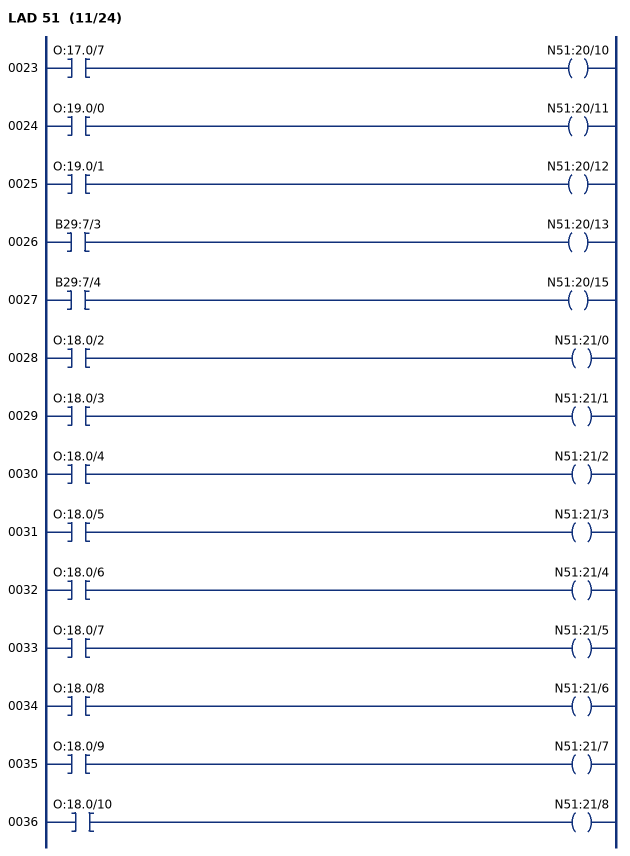
% Rung: 23 %
SOR XIC O:17.0/7 OTE N51:20/10 EOR
% Rung: 24 %
SOR XIC O:19.0/0 OTE N51:20/11 EOR
% Rung: 25 %
SOR XIC O:19.0/1 OTE N51:20/12 EOR
% Rung: 26 %
SOR XIC B29:7/3 OTE N51:20/13 EOR
% Rung: 27 %
SOR XIC B29:7/4 OTE N51:20/15 EOR
% Rung: 28 %
SOR XIC O:18.0/2 OTE N51:21/0 EOR
% Rung: 29 %
SOR XIC O:18.0/3 OTE N51:21/1 EOR
% Rung: 30 %
SOR XIC O:18.0/4 OTE N51:21/2 EOR
% Rung: 31 %
SOR XIC O:18.0/5 OTE N51:21/3 EOR
% Rung: 32 %
SOR XIC O:18.0/6 OTE N51:21/4 EOR
% Rung: 33 %
SOR XIC O:18.0/7 OTE N51:21/5 EOR
% Rung: 34 %
SOR XIC O:18.0/8 OTE N51:21/6 EOR
% Rung: 35 %
SOR XIC O:18.0/9 OTE N51:21/7 EOR
% Rung: 36 %
SOR XIC O:18.0/10 OTE N51:21/8 EOR

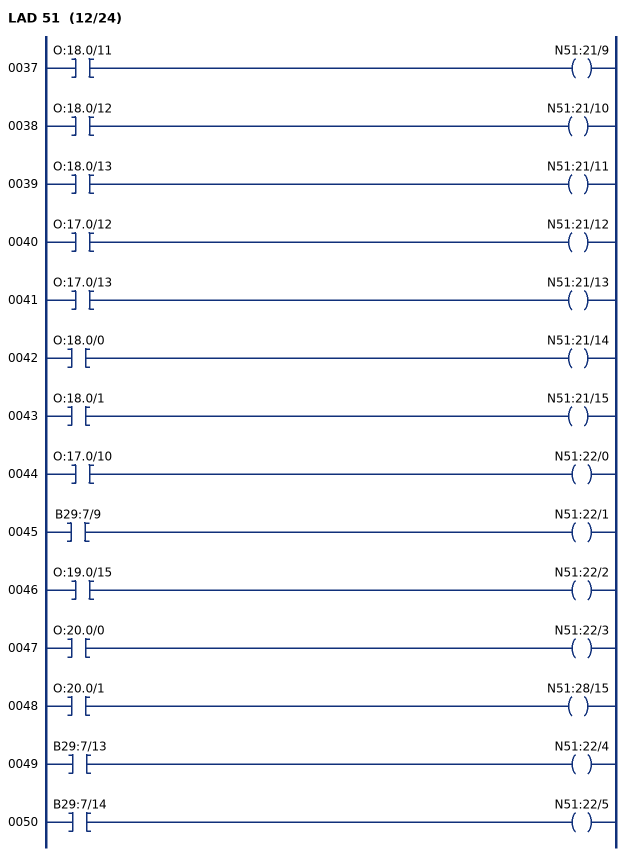
% Rung: 37 %
SOR XIC O:18.0/11 OTE N51:21/9 EOR
% Rung: 38 %
SOR XIC O:18.0/12 OTE N51:21/10 EOR
% Rung: 39 %
SOR XIC O:18.0/13 OTE N51:21/11 EOR
% Rung: 40 %
SOR XIC O:17.0/12 OTE N51:21/12 EOR
% Rung: 41 %
SOR XIC O:17.0/13 OTE N51:21/13 EOR
% Rung: 42 %
SOR XIC O:18.0/0 OTE N51:21/14 EOR
% Rung: 43 %
SOR XIC O:18.0/1 OTE N51:21/15 EOR
% Rung: 44 %
SOR XIC O:17.0/10 OTE N51:22/0 EOR
% Rung: 45 %
SOR XIC B29:7/9 OTE N51:22/1 EOR
% Rung: 46 %
SOR XIC O:19.0/15 OTE N51:22/2 EOR
% Rung: 47 %
SOR XIC O:20.0/0 OTE N51:22/3 EOR
% Rung: 48 %
SOR XIC O:20.0/1 OTE N51:28/15 EOR
% Rung: 49 %
SOR XIC B29:7/13 OTE N51:22/4 EOR
% Rung: 50 %
SOR XIC B29:7/14 OTE N51:22/5 EOR

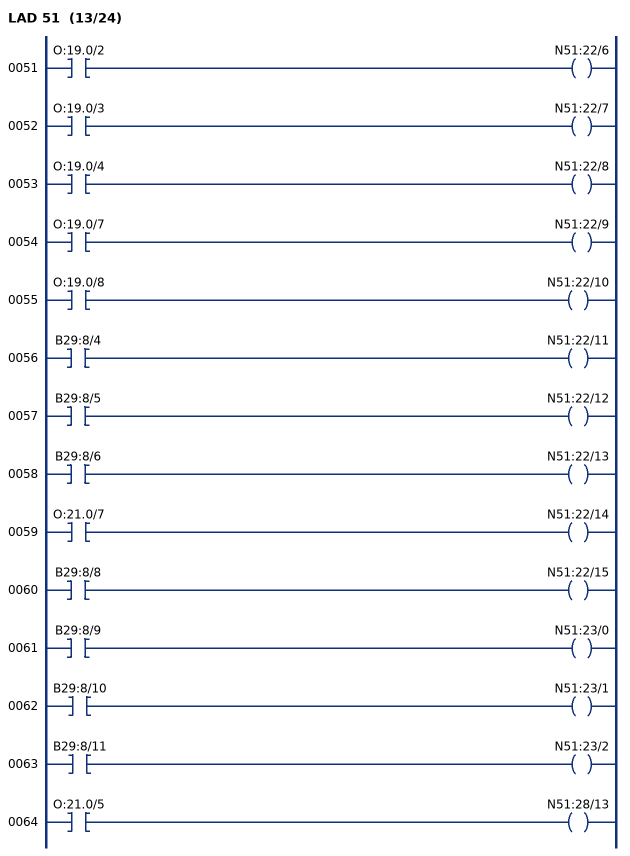
% Rung: 51 %
SOR XIC O:19.0/2 OTE N51:22/6 EOR
% Rung: 52 %
SOR XIC O:19.0/3 OTE N51:22/7 EOR
% Rung: 53 %
SOR XIC O:19.0/4 OTE N51:22/8 EOR
% Rung: 54 %
SOR XIC O:19.0/7 OTE N51:22/9 EOR
% Rung: 55 %
SOR XIC O:19.0/8 OTE N51:22/10 EOR
% Rung: 56 %
SOR XIC B29:8/4 OTE N51:22/11 EOR
% Rung: 57 %
SOR XIC B29:8/5 OTE N51:22/12 EOR
% Rung: 58 %
SOR XIC B29:8/6 OTE N51:22/13 EOR
% Rung: 59 %
SOR XIC O:21.0/7 OTE N51:22/14 EOR
% Rung: 60 %
SOR XIC B29:8/8 OTE N51:22/15 EOR
% Rung: 61 %
SOR XIC B29:8/9 OTE N51:23/0 EOR
% Rung: 62 %
SOR XIC B29:8/10 OTE N51:23/1 EOR
% Rung: 63 %
SOR XIC B29:8/11 OTE N51:23/2 EOR
% Rung: 64 %
SOR XIC O:21.0/5 OTE N51:28/13 EOR

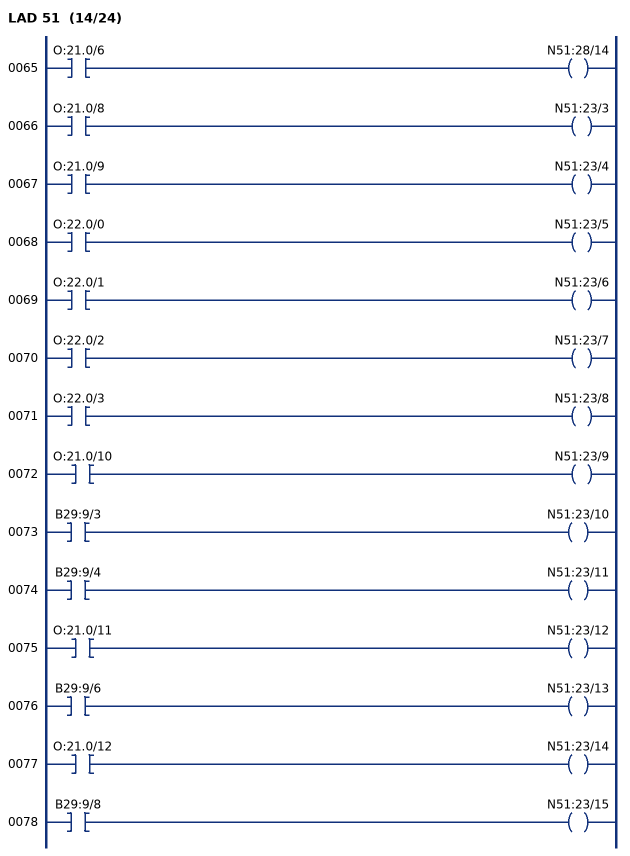
% Rung: 65 %
SOR XIC O:21.0/6 OTE N51:28/14 EOR
% Rung: 66 %
SOR XIC O:21.0/8 OTE N51:23/3 EOR
% Rung: 67 %
SOR XIC O:21.0/9 OTE N51:23/4 EOR
% Rung: 68 %
SOR XIC O:22.0/0 OTE N51:23/5 EOR
% Rung: 69 %
SOR XIC O:22.0/1 OTE N51:23/6 EOR
% Rung: 70 %
SOR XIC O:22.0/2 OTE N51:23/7 EOR
% Rung: 71 %
SOR XIC O:22.0/3 OTE N51:23/8 EOR
% Rung: 72 %
SOR XIC O:21.0/10 OTE N51:23/9 EOR
% Rung: 73 %
SOR XIC B29:9/3 OTE N51:23/10 EOR
% Rung: 74 %
SOR XIC B29:9/4 OTE N51:23/11 EOR
% Rung: 75 %
SOR XIC O:21.0/11 OTE N51:23/12 EOR
% Rung: 76 %
SOR XIC B29:9/6 OTE N51:23/13 EOR
% Rung: 77 %
SOR XIC O:21.0/12 OTE N51:23/14 EOR
% Rung: 78 %
SOR XIC B29:9/8 OTE N51:23/15 EOR

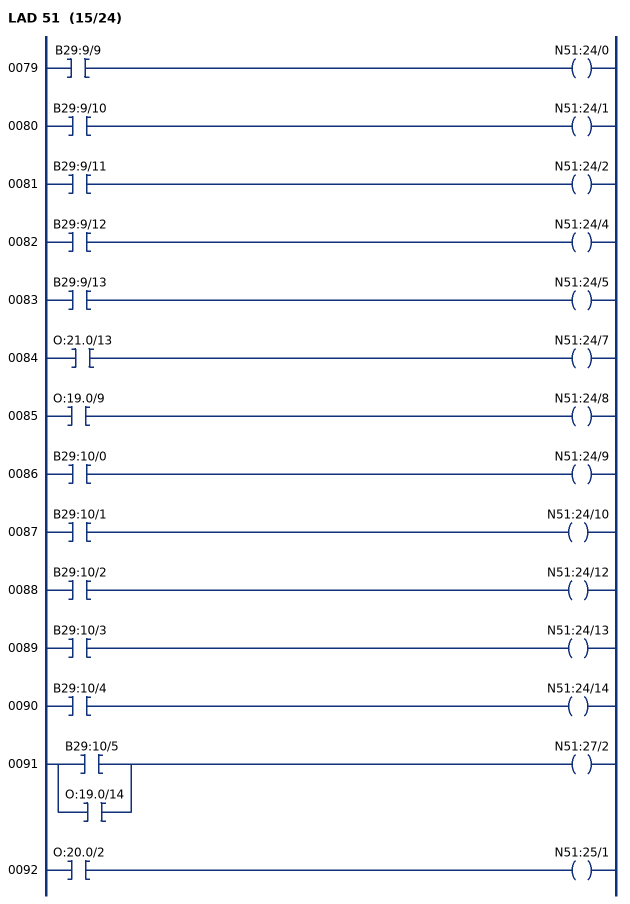
% Rung: 79 %
SOR XIC B29:9/9 OTE N51:24/0 EOR
% Rung: 80 %
SOR XIC B29:9/10 OTE N51:24/1 EOR
% Rung: 81 %
SOR XIC B29:9/11 OTE N51:24/2 EOR
% Rung: 82 %
SOR XIC B29:9/12 OTE N51:24/4 EOR
% Rung: 83 %
SOR XIC B29:9/13 OTE N51:24/5 EOR
% Rung: 84 %
SOR XIC O:21.0/13 OTE N51:24/7 EOR
% Rung: 85 %
SOR XIC O:19.0/9 OTE N51:24/8 EOR
% Rung: 86 %
SOR XIC B29:10/0 OTE N51:24/9 EOR
% Rung: 87 %
SOR XIC B29:10/1 OTE N51:24/10 EOR
% Rung: 88 %
SOR XIC B29:10/2 OTE N51:24/12 EOR
% Rung: 89 %
SOR XIC B29:10/3 OTE N51:24/13 EOR
% Rung: 90 %
SOR XIC B29:10/4 OTE N51:24/14 EOR
% Rung: 91 %
SOR BST XIC B29:10/5 NXB XIC O:19.0/14 BND OTE N51:27/2 EOR
% Rung: 92 %
SOR XIC O:20.0/2 OTE N51:25/1 EOR

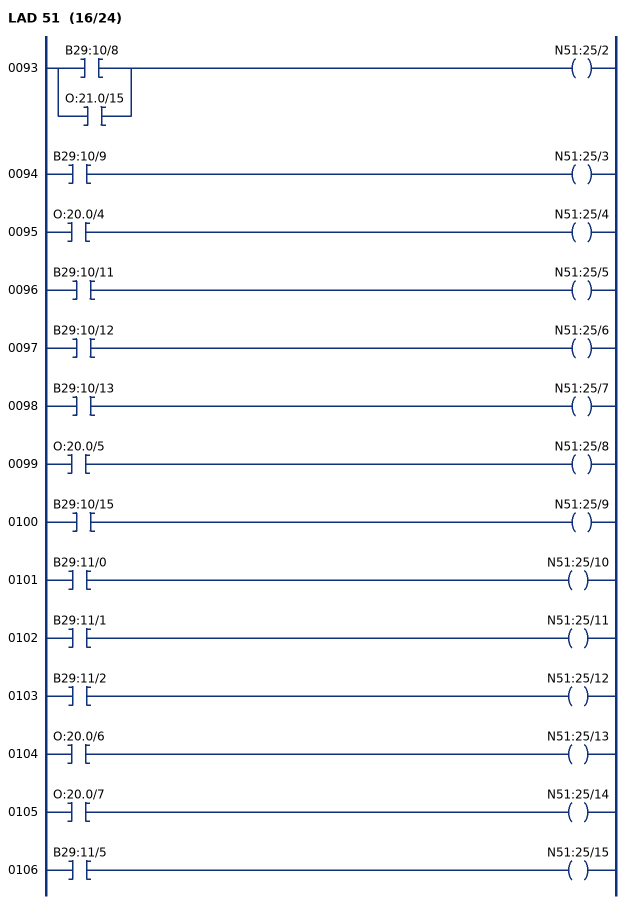
% Rung: 93 %
SOR BST XIC B29:10/8 NXB XIC O:21.0/15 BND OTE N51:25/2 EOR
% Rung: 94 %
SOR XIC B29:10/9 OTE N51:25/3 EOR
% Rung: 95 %
SOR XIC O:20.0/4 OTE N51:25/4 EOR
% Rung: 96 %
SOR XIC B29:10/11 OTE N51:25/5 EOR
% Rung: 97 %
SOR XIC B29:10/12 OTE N51:25/6 EOR
% Rung: 98 %
SOR XIC B29:10/13 OTE N51:25/7 EOR
% Rung: 99 %
SOR XIC O:20.0/5 OTE N51:25/8 EOR
% Rung: 100 %
SOR XIC B29:10/15 OTE N51:25/9 EOR
% Rung: 101 %
SOR XIC B29:11/0 OTE N51:25/10 EOR
% Rung: 102 %
SOR XIC B29:11/1 OTE N51:25/11 EOR
% Rung: 103 %
SOR XIC B29:11/2 OTE N51:25/12 EOR
% Rung: 104 %
SOR XIC O:20.0/6 OTE N51:25/13 EOR
% Rung: 105 %
SOR XIC O:20.0/7 OTE N51:25/14 EOR
% Rung: 106 %
SOR XIC B29:11/5 OTE N51:25/15 EOR

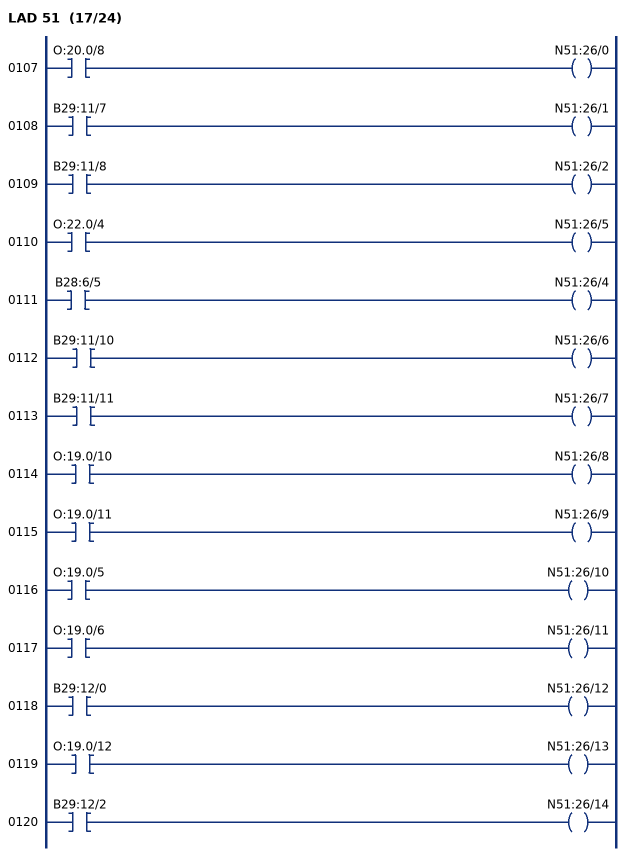
% Rung: 107 %
SOR XIC O:20.0/8 OTE N51:26/0 EOR
% Rung: 108 %
SOR XIC B29:11/7 OTE N51:26/1 EOR
% Rung: 109 %
SOR XIC B29:11/8 OTE N51:26/2 EOR
% Rung: 110 %
SOR XIC O:22.0/4 OTE N51:26/5 EOR
% Rung: 111 %
SOR XIC B28:6/5 OTE N51:26/4 EOR
% Rung: 112 %
SOR XIC B29:11/10 OTE N51:26/6 EOR
% Rung: 113 %
SOR XIC B29:11/11 OTE N51:26/7 EOR
% Rung: 114 %
SOR XIC O:19.0/10 OTE N51:26/8 EOR
% Rung: 115 %
SOR XIC O:19.0/11 OTE N51:26/9 EOR
% Rung: 116 %
SOR XIC O:19.0/5 OTE N51:26/10 EOR
% Rung: 117 %
SOR XIC O:19.0/6 OTE N51:26/11 EOR
% Rung: 118 %
SOR XIC B29:12/0 OTE N51:26/12 EOR
% Rung: 119 %
SOR XIC O:19.0/12 OTE N51:26/13 EOR
% Rung: 120 %
SOR XIC B29:12/2 OTE N51:26/14 EOR

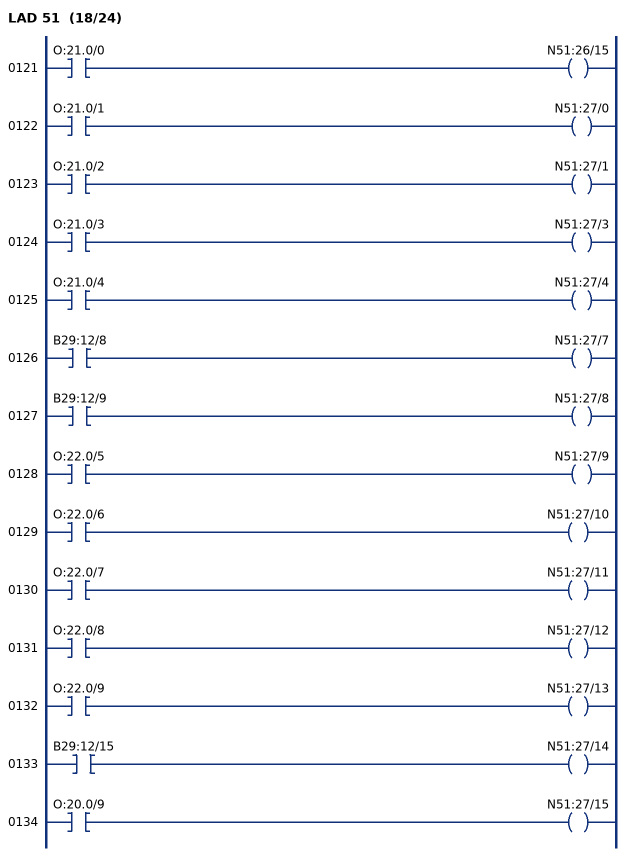
% Rung: 121 %
SOR XIC O:21.0/0 OTE N51:26/15 EOR
% Rung: 122 %
SOR XIC O:21.0/1 OTE N51:27/0 EOR
% Rung: 123 %
SOR XIC O:21.0/2 OTE N51:27/1 EOR
% Rung: 124 %
SOR XIC O:21.0/3 OTE N51:27/3 EOR
% Rung: 125 %
SOR XIC O:21.0/4 OTE N51:27/4 EOR
% Rung: 126 %
SOR XIC B29:12/8 OTE N51:27/7 EOR
% Rung: 127 %
SOR XIC B29:12/9 OTE N51:27/8 EOR
% Rung: 128 %
SOR XIC O:22.0/5 OTE N51:27/9 EOR
% Rung: 129 %
SOR XIC O:22.0/6 OTE N51:27/10 EOR
% Rung: 130 %
SOR XIC O:22.0/7 OTE N51:27/11 EOR
% Rung: 131 %
SOR XIC O:22.0/8 OTE N51:27/12 EOR
% Rung: 132 %
SOR XIC O:22.0/9 OTE N51:27/13 EOR
% Rung: 133 %
SOR XIC B29:12/15 OTE N51:27/14 EOR
% Rung: 134 %
SOR XIC O:20.0/9 OTE N51:27/15 EOR

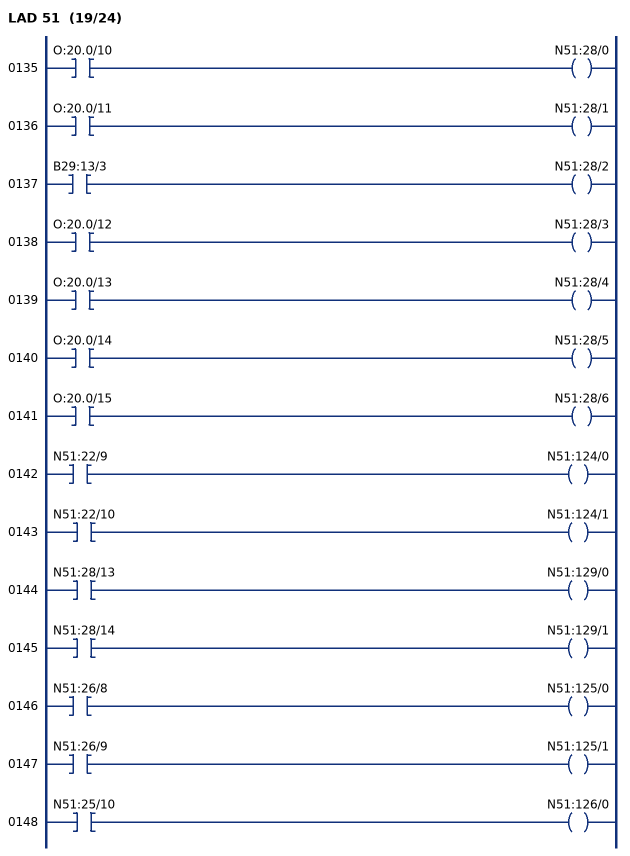
% Rung: 135 %
SOR XIC O:20.0/10 OTE N51:28/0 EOR
% Rung: 136 %
SOR XIC O:20.0/11 OTE N51:28/1 EOR
% Rung: 137 %
SOR XIC B29:13/3 OTE N51:28/2 EOR
% Rung: 138 %
SOR XIC O:20.0/12 OTE N51:28/3 EOR
% Rung: 139 %
SOR XIC O:20.0/13 OTE N51:28/4 EOR
% Rung: 140 %
SOR XIC O:20.0/14 OTE N51:28/5 EOR
% Rung: 141 %
SOR XIC O:20.0/15 OTE N51:28/6 EOR
% Rung: 142 %
SOR XIC N51:22/9 OTE N51:124/0 EOR
% Rung: 143 %
SOR XIC N51:22/10 OTE N51:124/1 EOR
% Rung: 144 %
SOR XIC N51:28/13 OTE N51:129/0 EOR
% Rung: 145 %
SOR XIC N51:28/14 OTE N51:129/1 EOR
% Rung: 146 %
SOR XIC N51:26/8 OTE N51:125/0 EOR
% Rung: 147 %
SOR XIC N51:26/9 OTE N51:125/1 EOR
% Rung: 148 %
SOR XIC N51:25/10 OTE N51:126/0 EOR

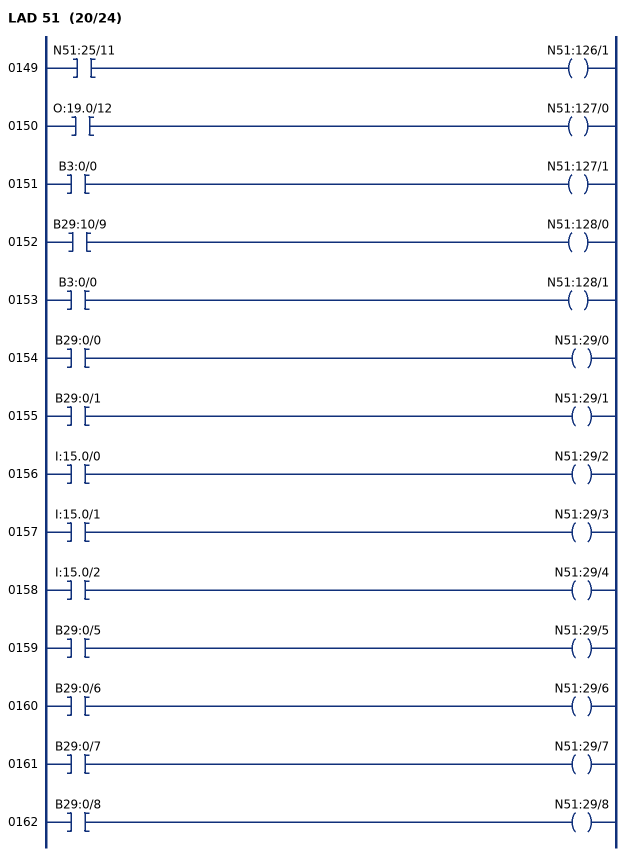
% Rung: 149 %
SOR XIC N51:25/11 OTE N51:126/1 EOR
% Rung: 150 %
SOR XIC O:19.0/12 OTE N51:127/0 EOR
% Rung: 151 %
SOR XIC B3:0/0 OTE N51:127/1 EOR
% Rung: 152 %
SOR XIC B29:10/9 OTE N51:128/0 EOR
% Rung: 153 %
SOR XIC B3:0/0 OTE N51:128/1 EOR
% Rung: 154 %
SOR XIC B29:0/0 OTE N51:29/0 EOR
% Rung: 155 %
SOR XIC B29:0/1 OTE N51:29/1 EOR
% Rung: 156 %
SOR XIC I:15.0/0 OTE N51:29/2 EOR
% Rung: 157 %
SOR XIC I:15.0/1 OTE N51:29/3 EOR
% Rung: 158 %
SOR XIC I:15.0/2 OTE N51:29/4 EOR
% Rung: 159 %
SOR XIC B29:0/5 OTE N51:29/5 EOR
% Rung: 160 %
SOR XIC B29:0/6 OTE N51:29/6 EOR
% Rung: 161 %
SOR XIC B29:0/7 OTE N51:29/7 EOR
% Rung: 162 %
SOR XIC B29:0/8 OTE N51:29/8 EOR

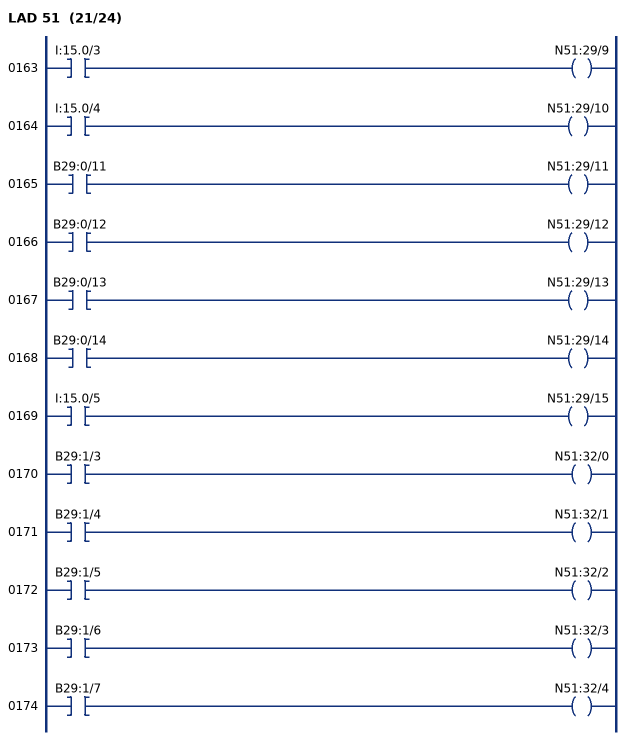
% Rung: 163 %
SOR XIC I:15.0/3 OTE N51:29/9 EOR
% Rung: 164 %
SOR XIC I:15.0/4 OTE N51:29/10 EOR
% Rung: 165 %
SOR XIC B29:0/11 OTE N51:29/11 EOR
% Rung: 166 %
SOR XIC B29:0/12 OTE N51:29/12 EOR
% Rung: 167 %
SOR XIC B29:0/13 OTE N51:29/13 EOR
% Rung: 168 %
SOR XIC B29:0/14 OTE N51:29/14 EOR
% Rung: 169 %
SOR XIC I:15.0/5 OTE N51:29/15 EOR
% Rung: 170 %
SOR XIC B29:1/3 OTE N51:32/0 EOR
% Rung: 171 %
SOR XIC B29:1/4 OTE N51:32/1 EOR
% Rung: 172 %
SOR XIC B29:1/5 OTE N51:32/2 EOR
% Rung: 173 %
SOR XIC B29:1/6 OTE N51:32/3 EOR
% Rung: 174 %
SOR XIC B29:1/7 OTE N51:32/4 EOR

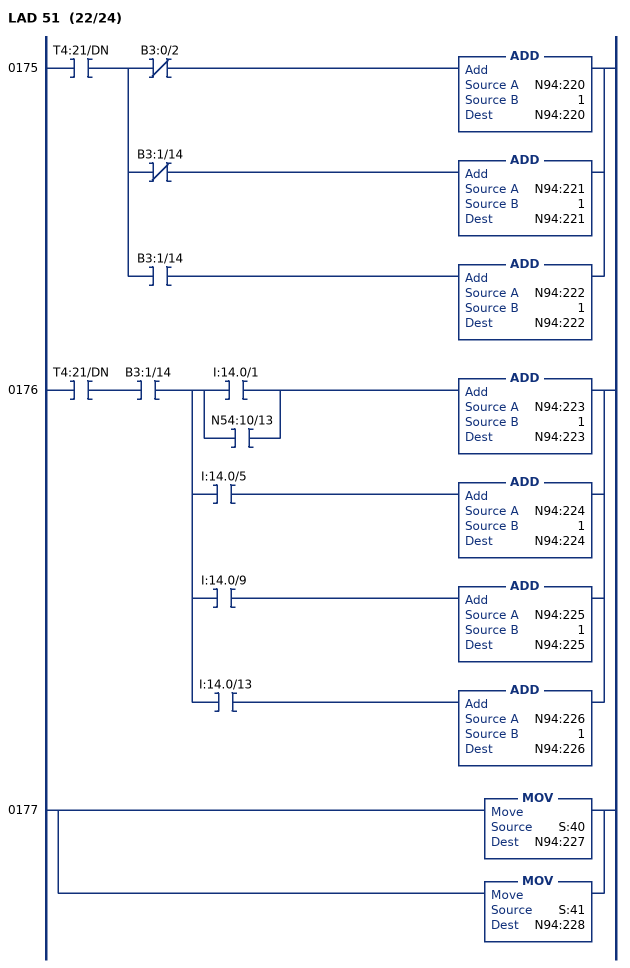
% Rung: 175 %
SOR XIC T4:21/DN BST XIO B3:0/2 ADD N94:220 1 N94:220 NXB XIO B3:1/14 ADD N94:221 1 N94:221 NXB XIC B3:1/14 ADD N94:222 1 N94:222 BND EOR
% Rung: 176 %
SOR XIC T4:21/DN XIC B3:1/14 BST BST XIC I:14.0/1 NXB XIC N54:10/13 BND ADD N94:223 1 N94:223 NXB XIC I:14.0/5 ADD N94:224 1 N94:224 NXB XIC I:14.0/9 ADD N94:225 1 N94:225 NXB XIC I:14.0/13 ADD N94:226 1 N94:226 BND EOR
% Rung: 177 %
SOR BST MOV S:40 N94:227 NXB MOV S:41 N94:228 BND EOR
%   S:40  "Clock Calendar Hours" %
%   S:41  "Clock Calendar Minutes" %

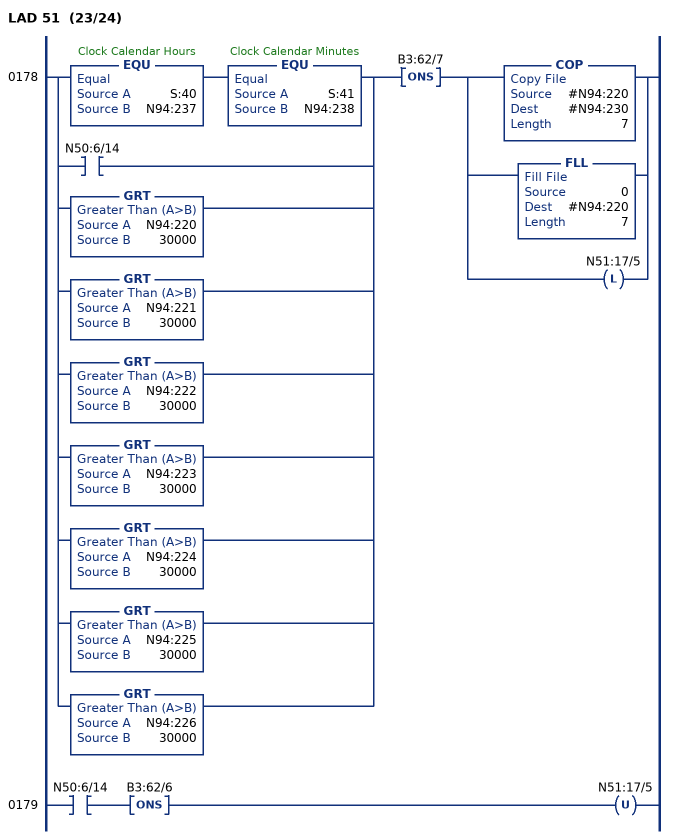
% Rung: 178 %
SOR BST EQU S:40 N94:237 EQU S:41 N94:238 NXB XIC N50:6/14 NXB GRT N94:220 30000 NXB GRT N94:221 30000 NXB GRT N94:222 30000 NXB GRT N94:223 30000 NXB GRT N94:224 30000 NXB GRT N94:225 30000 NXB GRT N94:226 30000 BND OSR B3:62/7 BST COP #N94:220 #N94:230 7 NXB FLL 0 #N94:220 7 NXB OTL N51:17/5 BND EOR
%   S:40  "Clock Calendar Hours" %
%   S:41  "Clock Calendar Minutes" %
% Rung: 179 %
SOR XIC N50:6/14 OSR B3:62/6 OTU N51:17/5 EOR

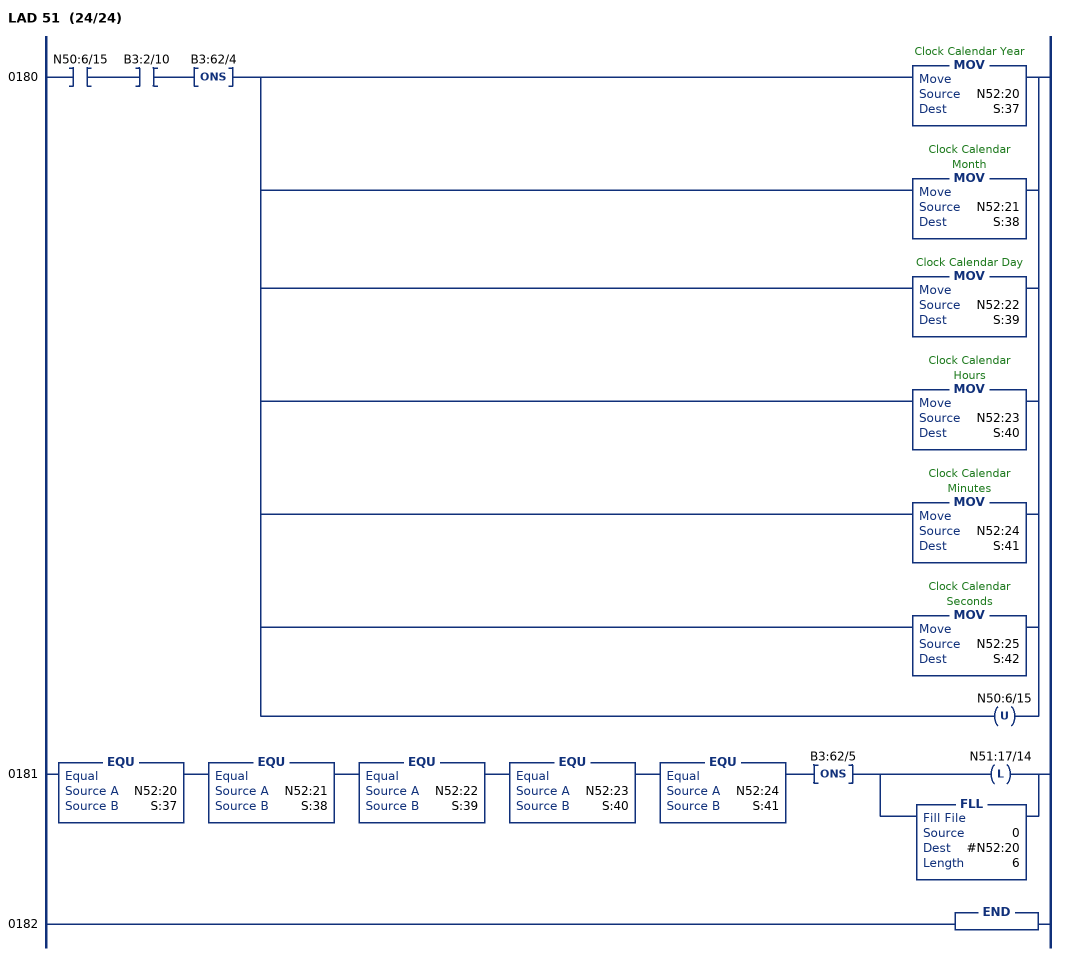
% Rung: 180 %
SOR XIC N50:6/15 XIC B3:2/10 OSR B3:62/4 BST MOV N52:20 S:37 NXB MOV N52:21 S:38 NXB MOV N52:22 S:39 NXB MOV N52:23 S:40 NXB MOV N52:24 S:41 NXB MOV N52:25 S:42 NXB OTU N50:6/15 BND EOR
%   S:37  "Clock Calendar Year" %
%   S:38  "Clock Calendar Month" %
%   S:39  "Clock Calendar Day" %
%   S:40  "Clock Calendar Hours" %
%   S:41  "Clock Calendar Minutes" %
%   S:42  "Clock Calendar Seconds" %
% Rung: 181 %
SOR EQU N52:20 S:37 EQU N52:21 S:38 EQU N52:22 S:39 EQU N52:23 S:40 EQU N52:24 S:41 OSR B3:62/5 BST OTL N51:17/14 NXB FLL 0 #N52:20 6 BND EOR
%   S:37  "Clock Calendar Year" %
%   S:38  "Clock Calendar Month" %
%   S:39  "Clock Calendar Day" %
%   S:40  "Clock Calendar Hours" %
%   S:41  "Clock Calendar Minutes" %
% Rung: 182 %
SOR END EOR

LADDER 52
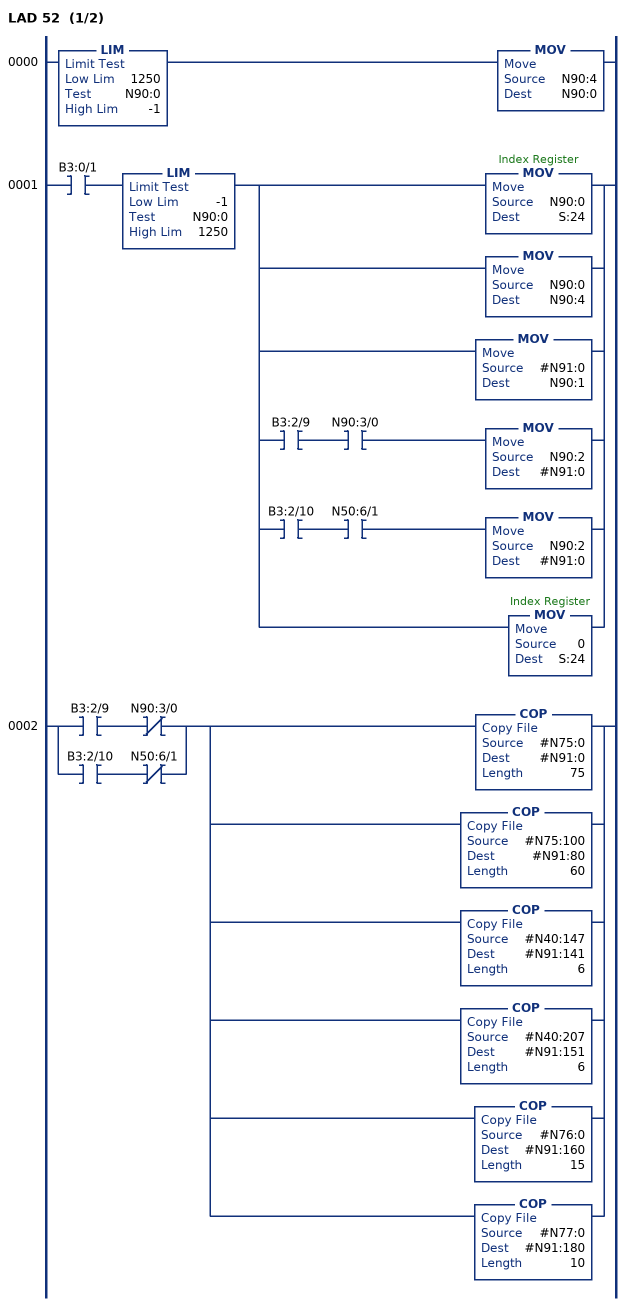
% Rung: 0 %
SOR LIM 1250 N90:0 -1 MOV N90:4 N90:0 EOR
% Rung: 1 %
SOR XIC B3:0/1 LIM -1 N90:0 1250 BST MOV N90:0 S:24 NXB MOV N90:0 N90:4 NXB MOV #N91:0 N90:1 NXB XIC B3:2/9 XIC N90:3/0 MOV N90:2 #N91:0 NXB XIC B3:2/10 XIC N50:6/1 MOV N90:2 #N91:0 NXB MOV 0 S:24 BND EOR
%   S:24  "Index Register" %
% Rung: 2 %
SOR BST XIC B3:2/9 XIO N90:3/0 NXB XIC B3:2/10 XIO N50:6/1 BND BST COP #N75:0 #N91:0 75 NXB COP #N75:100 #N91:80 60 NXB COP #N40:147 #N91:141 6 NXB COP #N40:207 #N91:151 6 NXB COP #N76:0 #N91:160 15 NXB COP #N77:0 #N91:180 10 BND EOR

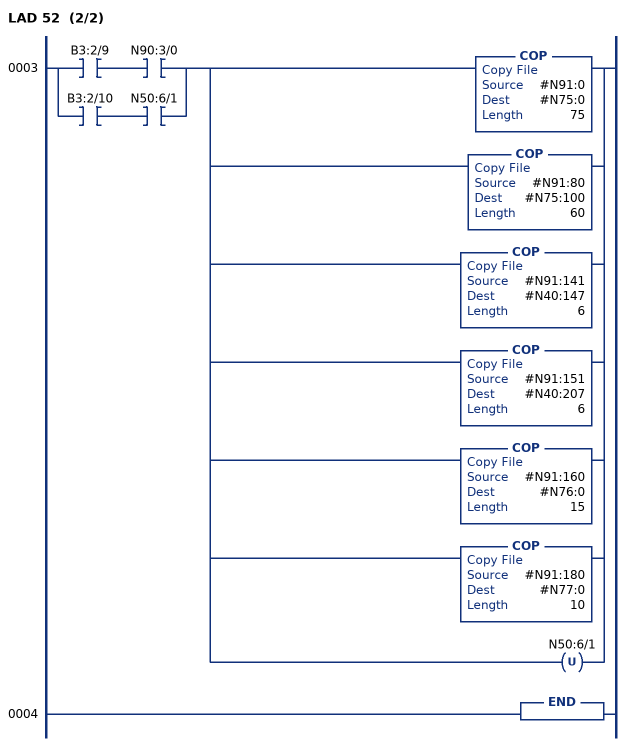
% Rung: 3 %
SOR BST XIC B3:2/9 XIC N90:3/0 NXB XIC B3:2/10 XIC N50:6/1 BND BST COP #N91:0 #N75:0 75 NXB COP #N91:80 #N75:100 60 NXB COP #N91:141 #N40:147 6 NXB COP #N91:151 #N40:207 6 NXB COP #N91:160 #N76:0 15 NXB COP #N91:180 #N77:0 10 NXB OTU N50:6/1 BND EOR
% Rung: 4 %
SOR END EOR

LADDER 53
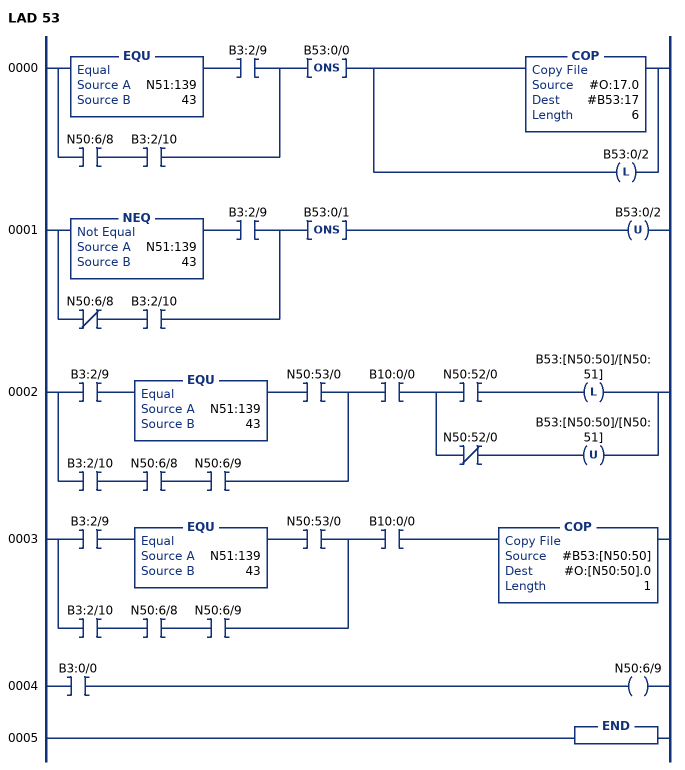
% Rung: 0 %
SOR BST EQU N51:139 43 XIC B3:2/9 NXB XIC N50:6/8 XIC B3:2/10 BND OSR B53:0/0 BST COP #O:17.0 #B53:17 6 NXB OTL B53:0/2 BND EOR
% Rung: 1 %
SOR BST NEQ N51:139 43 XIC B3:2/9 NXB XIO N50:6/8 XIC B3:2/10 BND OSR B53:0/1 OTU B53:0/2 EOR
% Rung: 2 %
SOR BST XIC B3:2/9 EQU N51:139 43 XIC N50:53/0 NXB XIC B3:2/10 XIC N50:6/8 XIC N50:6/9 BND XIC B10:0/0 BST XIC N50:52/0 OTL B53:[N50:50]/[N50:51] NXB XIO N50:52/0 OTU B53:[N50:50]/[N50:51] BND EOR
% Rung: 3 %
SOR BST XIC B3:2/9 EQU N51:139 43 XIC N50:53/0 NXB XIC B3:2/10 XIC N50:6/8 XIC N50:6/9 BND XIC B10:0/0 COP #B53:[N50:50] #O:[N50:50].0 1 EOR
% Rung: 4 %
SOR XIC B3:0/0 OTE N50:6/9 EOR
% Rung: 5 %
SOR END EOR

LADDER 60
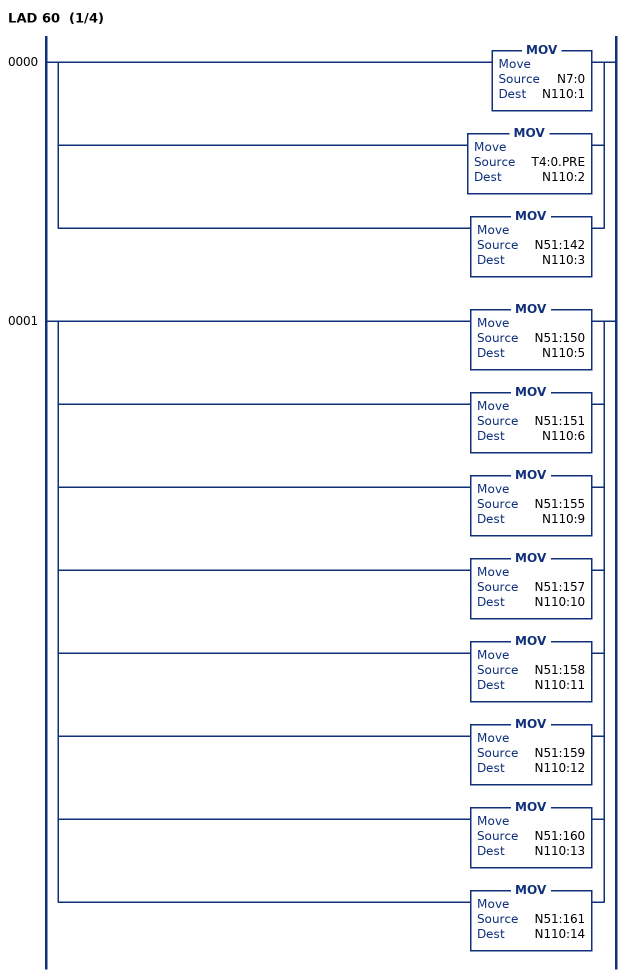
% Rung: 0 %
SOR BST MOV N7:0 N110:1 NXB MOV T4:0.PRE N110:2 NXB MOV N51:142 N110:3 BND EOR
% Rung: 1 %
SOR BST MOV N51:150 N110:5 NXB MOV N51:151 N110:6 NXB MOV N51:155 N110:9 NXB MOV N51:157 N110:10 NXB MOV N51:158 N110:11 NXB MOV N51:159 N110:12 NXB MOV N51:160 N110:13 NXB MOV N51:161 N110:14 BND EOR

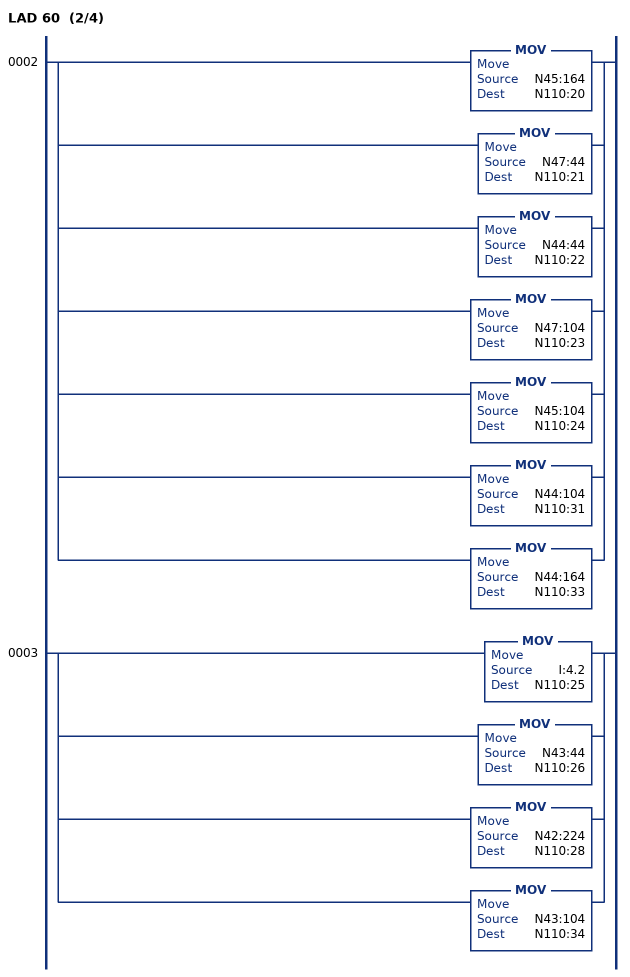
% Rung: 2 %
SOR BST MOV N45:164 N110:20 NXB MOV N47:44 N110:21 NXB MOV N44:44 N110:22 NXB MOV N47:104 N110:23 NXB MOV N45:104 N110:24 NXB MOV N44:104 N110:31 NXB MOV N44:164 N110:33 BND EOR
% Rung: 3 %
SOR BST MOV I:4.2 N110:25 NXB MOV N43:44 N110:26 NXB MOV N42:224 N110:28 NXB MOV N43:104 N110:34 BND EOR

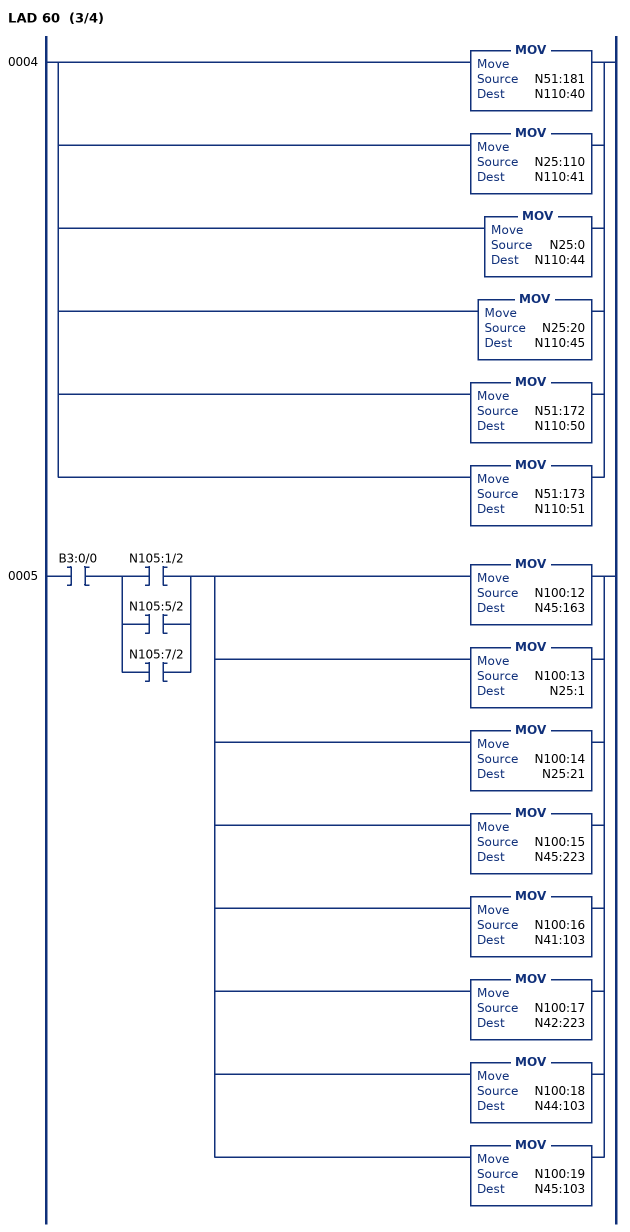
% Rung: 4 %
SOR BST MOV N51:181 N110:40 NXB MOV N25:110 N110:41 NXB MOV N25:0 N110:44 NXB MOV N25:20 N110:45 NXB MOV N51:172 N110:50 NXB MOV N51:173 N110:51 BND EOR
% Rung: 5 %
SOR XIC B3:0/0 BST XIC N105:1/2 NXB XIC N105:5/2 NXB XIC N105:7/2 BND BST MOV N100:12 N45:163 NXB MOV N100:13 N25:1 NXB MOV N100:14 N25:21 NXB MOV N100:15 N45:223 NXB MOV N100:16 N41:103 NXB MOV N100:17 N42:223 NXB MOV N100:18 N44:103 NXB MOV N100:19 N45:103 BND EOR

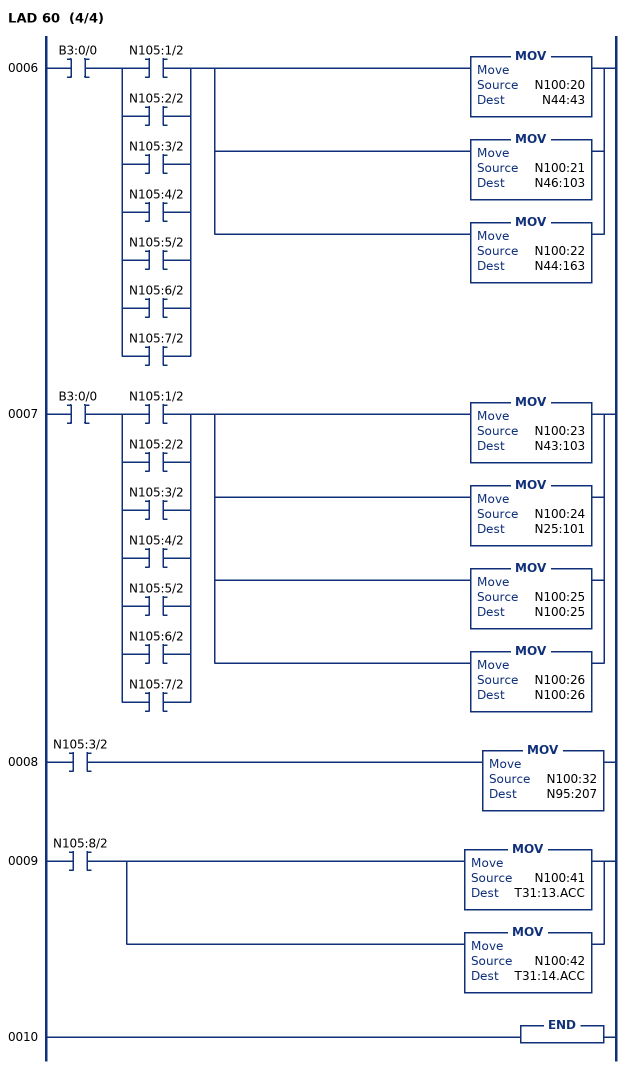
% Rung: 6 %
SOR XIC B3:0/0 BST XIC N105:1/2 NXB XIC N105:2/2 NXB XIC N105:3/2 NXB XIC N105:4/2 NXB XIC N105:5/2 NXB XIC N105:6/2 NXB XIC N105:7/2 BND BST MOV N100:20 N44:43 NXB MOV N100:21 N46:103 NXB MOV N100:22 N44:163 BND EOR
% Rung: 7 %
SOR XIC B3:0/0 BST XIC N105:1/2 NXB XIC N105:2/2 NXB XIC N105:3/2 NXB XIC N105:4/2 NXB XIC N105:5/2 NXB XIC N105:6/2 NXB XIC N105:7/2 BND BST MOV N100:23 N43:103 NXB MOV N100:24 N25:101 NXB MOV N100:25 N100:25 NXB MOV N100:26 N100:26 BND EOR
% Rung: 8 %
SOR XIC N105:3/2 MOV N100:32 N95:207 EOR
% Rung: 9 %
SOR XIC N105:8/2 BST MOV N100:41 T31:13.ACC NXB MOV N100:42 T31:14.ACC BND EOR
% Rung: 10 %
SOR END EOR

LADDER 71
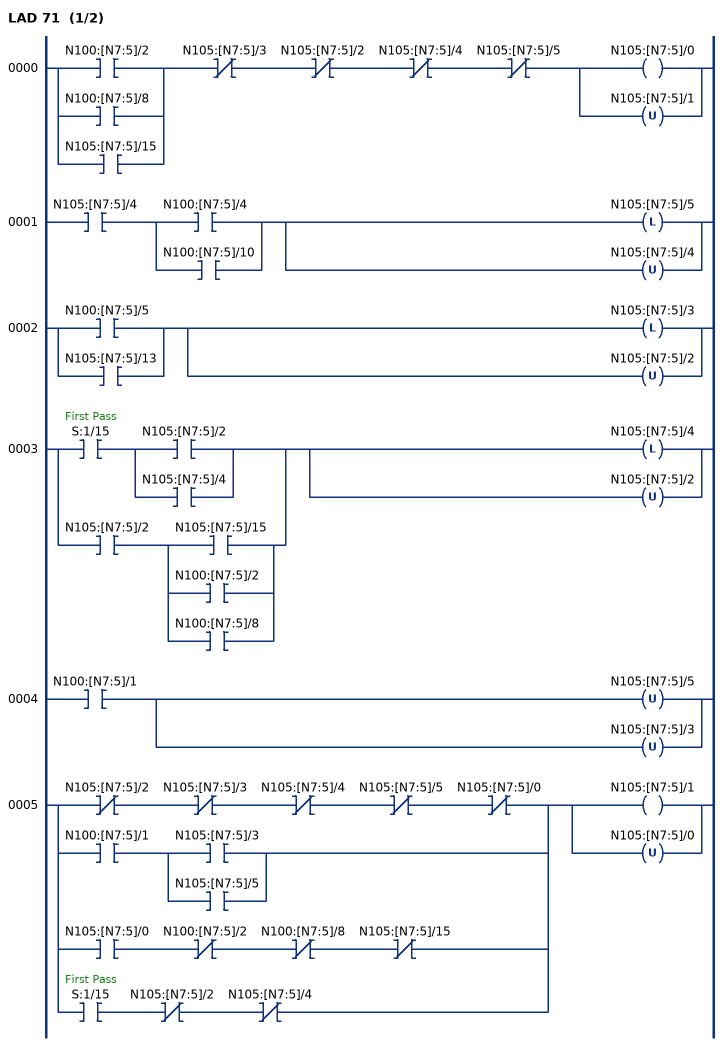
% Rung: 0 %
SOR BST XIC N100:[N7:5]/2 NXB XIC N100:[N7:5]/8 NXB XIC N105:[N7:5]/15 BND XIO N105:[N7:5]/3 XIO N105:[N7:5]/2 XIO N105:[N7:5]/4 XIO N105:[N7:5]/5 BST OTE N105:[N7:5]/0 NXB OTU N105:[N7:5]/1 BND EOR
% Rung: 1 %
SOR XIC N105:[N7:5]/4 BST XIC N100:[N7:5]/4 NXB XIC N100:[N7:5]/10 BND BST OTL N105:[N7:5]/5 NXB OTU N105:[N7:5]/4 BND EOR
% Rung: 2 %
SOR BST XIC N100:[N7:5]/5 NXB XIC N105:[N7:5]/13 BND BST OTL N105:[N7:5]/3 NXB OTU N105:[N7:5]/2 BND EOR
% Rung: 3 %
SOR BST XIC S:1/15 BST XIC N105:[N7:5]/2 NXB XIC N105:[N7:5]/4 BND NXB XIC N105:[N7:5]/2 BST XIC N105:[N7:5]/15 NXB XIC N100:[N7:5]/2 NXB XIC N100:[N7:5]/8 BND BND BST OTL N105:[N7:5]/4 NXB OTU N105:[N7:5]/2 BND EOR
%   S:1/15  "First Pass" %
% Rung: 4 %
SOR XIC N100:[N7:5]/1 BST OTU N105:[N7:5]/5 NXB OTU N105:[N7:5]/3 BND EOR
% Rung: 5 %
SOR BST XIO N105:[N7:5]/2 XIO N105:[N7:5]/3 XIO N105:[N7:5]/4 XIO N105:[N7:5]/5 XIO N105:[N7:5]/0 NXB XIC N100:[N7:5]/1 BST XIC N105:[N7:5]/3 NXB XIC N105:[N7:5]/5 BND NXB XIC N105:[N7:5]/0 XIO N100:[N7:5]/2 XIO N100:[N7:5]/8 XIO N105:[N7:5]/15 NXB XIC S:1/15 XIO N105:[N7:5]/2 XIO N105:[N7:5]/4 BND BST OTE N105:[N7:5]/1 NXB OTU N105:[N7:5]/0 BND EOR
%   S:1/15  "First Pass" %

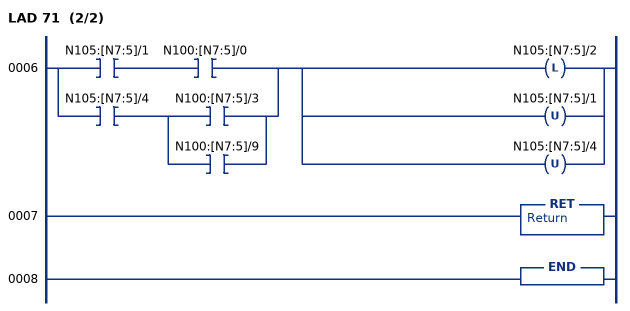
% Rung: 6 %
SOR BST XIC N105:[N7:5]/1 XIC N100:[N7:5]/0 NXB XIC N105:[N7:5]/4 BST XIC N100:[N7:5]/3 NXB XIC N100:[N7:5]/9 BND BND BST OTL N105:[N7:5]/2 NXB OTU N105:[N7:5]/1 NXB OTU N105:[N7:5]/4 BND EOR
% Rung: 7 %
SOR RET EOR
% Rung: 8 %
SOR END EOR

LADDER 75
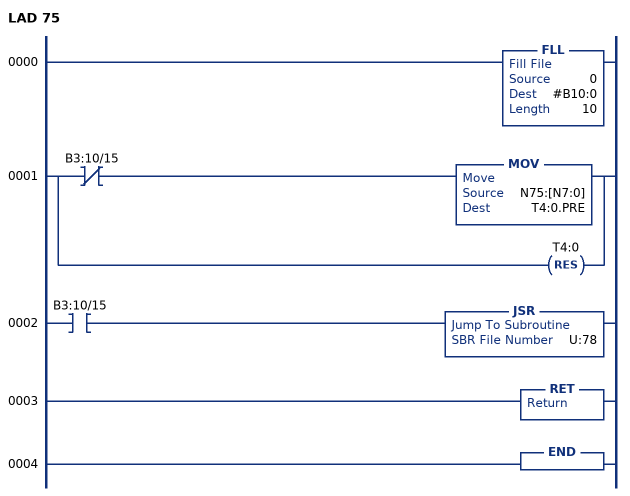
% Rung: 0 %
SOR FLL 0 #B10:0 10 EOR
% Rung: 1 %
SOR BST XIO B3:10/15 MOV N75:[N7:0] T4:0.PRE NXB RES T4:0 BND EOR
% Rung: 2 %
SOR XIC B3:10/15 JSR U:78 EOR
% Rung: 3 %
SOR RET EOR
% Rung: 4 %
SOR END EOR

LADDER 76
